# EPICS substitutions: multicastTestApp/Db/userHost.substitutions
# Example substitutions file

file "db/dbExample1.db" {
    { user = "tomytsaiHost" }
}

file db/dbExample2.db {
    pattern { user, no, scan }
        { "tomytsaiHost", 1, "1 second" }
        { "tomytsaiHost", 2, "2 second" }
        { "tomytsaiHost", 3, "5 second" }
}
